PROGRAM Systemparameter
VAR
END_VAR

// Lesen
	// Objektzustände
	GVL.Robot_State 		:= Anlage.UR5.P_State;
	GVL.Greifer_State 		:= Anlage.Gripper.P_State;
	GVL.Sensor_State 		:= Anlage.HEX_E.P_State;

// Zuweisen
	// Eigenschaften	
	Anlage.HEX_E.P_LimitValue 		:= GVL.eKraftLimitValue;
	Anlage.HEX_E.P_ErreichtValue 	:= GVL.eKraftErreichtValue

END_PROGRAM

(* stored: Version 1.1.0.1
   POU Systemparameter: Id {d577e6da-3909-4d5f-9dd0-cda923279a4c}, SpecialFunc None *)
